// TIA Portal V18 program export: 1 tag tables, 0 data types, 1 data blocks, 7 code blocks (in call order from the OBs), 5 instance data blocks

VAR_GLOBAL   // PLC tag table "Default tag table"
   "Motor start" AT %I0.0 : Bool;
   "Motor Stop" AT %I0.1 : Bool;
   Tag_2 AT %I0.2 : Bool;
   Tag_4 AT %I0.3 : Bool;
   "Motor running LED" AT %Q0.0 : Bool;
   "Motor contactor" AT %Q0.2 : Bool;
   Tag_1 AT %M10.0 : Bool;
   Tag_3 AT %M10.1 : Bool;
   System_Byte AT %MB88 : Byte;
   FirstScan AT %M88.0 : Bool;
   DiagStatusUpdate AT %M88.1 : Bool;
   AlwaysTRUE AT %M88.2 : Bool;
   AlwaysFALSE AT %M88.3 : Bool;
   "System_Byte(1)" AT %MB88 : Byte;
   Clock_Byte AT %MB0 : Byte;
   Clock_10Hz AT %M0.0 : Bool;
   Clock_5Hz AT %M0.1 : Bool;
   "Clock_2.5Hz" AT %M0.2 : Bool;
   Clock_2Hz AT %M0.3 : Bool;
   "Clock_1.25Hz" AT %M0.4 : Bool;
   Clock_1Hz AT %M0.5 : Bool;
   "Clock_0.625Hz" AT %M0.6 : Bool;
   "Clock_0.5Hz" AT %M0.7 : Bool;
   Alarm AT %MW40 : Word;
   Tag_5 AT %M40.0 : Bool;
END_VAR

DATA_BLOCK "Global data"   // DB2
{ S7_Optimized_Access := 'TRUE' }
VERSION : 0.1
// stored: AutoNumber true, DBAccessibleFromOPCUA true, IsOnlyStoredInLoadMemory false, IsRetainMemResEnabled false, IsWriteProtectedInAS false, MemoryReserve 100
   VAR
      data1 : Bool;
      data2 : Bool;
      data3 : Bool;
      data4 : Bool;
      data5 : Bool;
      data6 : Bool;
      data7 : Bool;
      data8 : Bool;
   END_VAR
   VAR RETAIN
      dataB1 : Byte := 10;
   END_VAR
   VAR
      dataB2 : Byte := 10;
      dataB3 : Byte := 10;
      dataB4 : Byte := 10;
      dataW1 : Word := 10;
   END_VAR
   VAR RETAIN
      dataW2 : Word := 20;
      dataW3 : Word := 20;
      dataW4 : Word := 20;
   END_VAR
   VAR
      dataW5 : Word := 20;
   END_VAR
BEGIN
END_DATA_BLOCK

ORGANIZATION_BLOCK "Main"   // OB1, LAD, ProgramCycle
TITLE = "Main Program Sweep (Cycle)"
{ S7_Optimized_Access := 'TRUE' }
VERSION : 0.1
// stored: AutoNumber true, IsIECCheckEnabled false, SetENOAutomatically false
   VAR_INPUT
      Initial_Call : Bool;   // Initial call of this OB
      Remanence : Bool;   // =True, if remanent data are available
   END_VAR
BEGIN

REGION Network 1
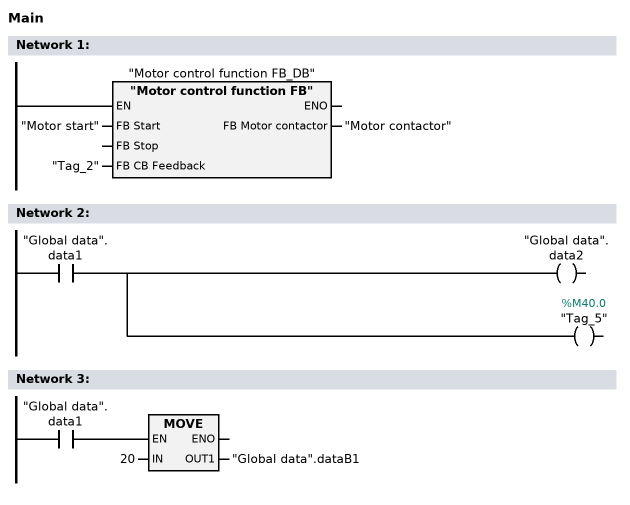
   RUNG wire#powerrail
      "Motor control function FB_DB"("FB Start" := "Motor start", "FB Stop" :=, "FB CB Feedback" := "Tag_2", "FB Motor contactor" => "Motor contactor")
   END_RUNG
   // the same network as SCL:
   "Motor control function FB_DB"("FB Start" := "Motor start",   // "Motor control function FB"
                           "FB CB Feedback" := "Tag_2",
                           "FB Motor contactor" => "Motor contactor");
END_REGION

REGION Network 2
   RUNG wire#powerrail
      Contact( "Global data".data1 )
      wire#w1
      Coil( "Global data".data2 )
   END_RUNG
   RUNG wire#w1
      Coil( "Tag_5" )
   END_RUNG
   // the same network as SCL:
   "Global data".data2 := "Global data".data1;
   "Tag_5" := "Global data".data1;
END_REGION

REGION Network 3
   RUNG wire#powerrail
      Contact( "Global data".data1 )
      Move(in := 20, out1 => "Global data".dataB1)
   END_RUNG
   // the same network as SCL:
   IF "Global data".data1 THEN "Global data".dataB1 := 20; END_IF;
END_REGION
END_ORGANIZATION_BLOCK

FUNCTION_BLOCK "Motor control function FB"   // FB1, LAD
{ S7_Optimized_Access := 'TRUE' }
VERSION : 0.1
// stored: AutoNumber true, IsIECCheckEnabled false, IsRetainMemResEnabled false, MemoryReserve 100, SetENOAutomatically false, UDAEnableTagReadback false
   VAR_INPUT
      "FB Start" : Bool;
      "FB Stop" : Bool;
      "FB CB Feedback" : Bool;
   END_VAR
   VAR_OUTPUT
      "FB Motor contactor" : Bool;
   END_VAR
BEGIN

REGION Network 1: Start motor contactor
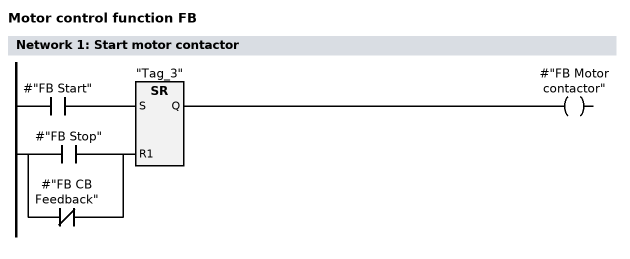
   RUNG wire#powerrail
      Contact( #"FB Start" )
      S_SR(operand := "Tag_3", r1 := wire#w1)
      Coil( #"FB Motor contactor" )
   END_RUNG
   RUNG wire#powerrail
      Contact( #"FB Stop" )
   END_RUNG wire#w1
   RUNG wire#powerrail
      I_Contact( #"FB CB Feedback" )
   END_RUNG wire#w1
   // the same network as SCL:
   IF #"FB Start" THEN
       "Tag_3" := TRUE;   // SR flip-flop
   END_IF;
   IF #"FB Stop" OR NOT #"FB CB Feedback" THEN "Tag_3" := FALSE; END_IF;
   #"FB Motor contactor" := "Tag_3";
END_REGION
END_FUNCTION_BLOCK

FUNCTION "Motor control Function FC" : Void   // FC2, LAD
{ S7_Optimized_Access := 'TRUE' }
VERSION : 0.1
// stored: AutoNumber true, IsIECCheckEnabled false, SetENOAutomatically false, UDAEnableTagReadback false
   VAR_INPUT
      Start : Bool;   // Input to start motor
      Stop : Bool;   // input to stop motor
      "CB feedback" : Bool;
   END_VAR
   VAR_OUTPUT
      "Motor contactor" : Bool;   // Start motor contactor
   END_VAR
BEGIN

REGION Network 1: Start motor contactor
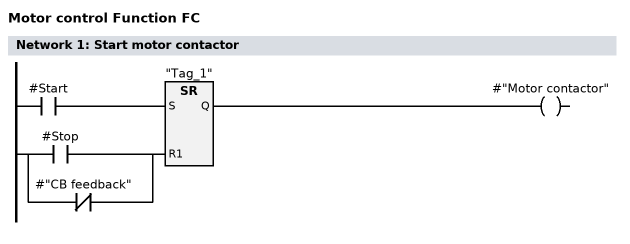
   RUNG wire#powerrail
      Contact( #Start )
      S_SR(operand := "Tag_1", r1 := wire#w1)
      Coil( #"Motor contactor" )
   END_RUNG
   RUNG wire#powerrail
      Contact( #Stop )
   END_RUNG wire#w1
   RUNG wire#powerrail
      I_Contact( #"CB feedback" )
   END_RUNG wire#w1
   // the same network as SCL:
   IF #Start THEN
       "Tag_1" := TRUE;   // SR flip-flop
   END_IF;
   IF #Stop OR NOT #"CB feedback" THEN "Tag_1" := FALSE; END_IF;
   #"Motor contactor" := "Tag_1";
END_REGION
END_FUNCTION

FUNCTION "Motor_control_FC" : Void   // FC1, LAD
{ S7_Optimized_Access := 'TRUE' }
VERSION : 0.1
// stored: AutoNumber true, IsIECCheckEnabled false, SetENOAutomatically false, UDAEnableTagReadback false
BEGIN

REGION Network 1
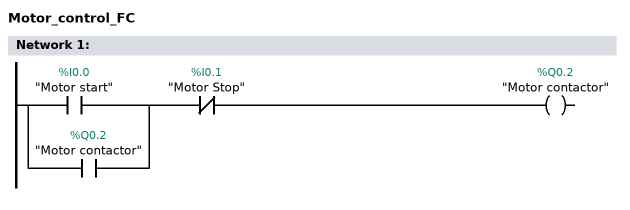
   RUNG wire#powerrail
      Contact( "Motor start" )
      wire#w1
      I_Contact( "Motor Stop" )
      Coil( "Motor contactor" )
   END_RUNG
   RUNG wire#powerrail
      Contact( "Motor contactor" )
   END_RUNG wire#w1
   // the same network as SCL:
   "Motor contactor" := ("Motor start" OR "Motor contactor") AND NOT "Motor Stop";
END_REGION
END_FUNCTION

FUNCTION_BLOCK "Multi instance FB"   // FB2, LAD
{ S7_Optimized_Access := 'TRUE' }
VERSION : 0.1
// stored: AutoNumber true, IsIECCheckEnabled false, IsRetainMemResEnabled false, MemoryReserve 100, SetENOAutomatically false, UDAEnableTagReadback false
   VAR
      "Motor control function FB_Instance" { S7_SetPoint := 'True'} : "Motor control function FB";
      "Motor control function FB_Instance_1" { S7_SetPoint := 'True'} : "Motor control function FB";
   END_VAR
BEGIN

REGION Network 1: Motor 1
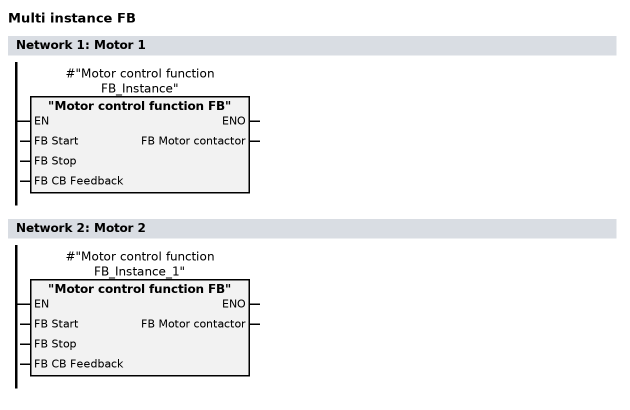
   RUNG wire#powerrail
      #"Motor control function FB_Instance"("FB Start" :=, "FB Stop" :=, "FB CB Feedback" :=, "FB Motor contactor" =>)
   END_RUNG
   // the same network as SCL:
   #"Motor control function FB_Instance"();   // "Motor control function FB"
END_REGION

REGION Network 2: Motor 2
   RUNG wire#powerrail
      #"Motor control function FB_Instance_1"("FB Start" :=, "FB Stop" :=, "FB CB Feedback" :=, "FB Motor contactor" =>)
   END_RUNG
   // the same network as SCL:
   #"Motor control function FB_Instance_1"();   // "Motor control function FB"
END_REGION
END_FUNCTION_BLOCK

FUNCTION "Sunc_2" : Void   // FC4, LAD
{ S7_Optimized_Access := 'TRUE' }
VERSION : 0.1
// stored: AutoNumber true, IsIECCheckEnabled false, SetENOAutomatically false, UDAEnableTagReadback false
BEGIN

REGION Network 1
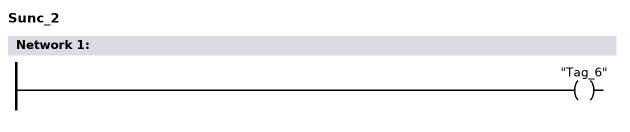
   RUNG wire#powerrail
      Coil( "Tag_6" )
   END_RUNG
   // the same network as SCL:
   "Tag_6" := TRUE;
END_REGION
END_FUNCTION

FUNCTION "Sync_Test" : Void   // FC3, LAD
{ S7_Optimized_Access := 'TRUE' }
VERSION : 0.1
// stored: AutoNumber true, IsIECCheckEnabled false, SetENOAutomatically false, UDAEnableTagReadback false
BEGIN

REGION Network 1
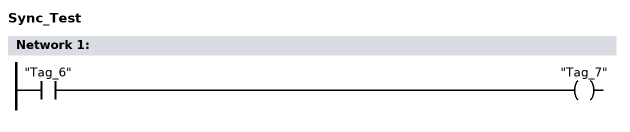
   RUNG wire#powerrail
      Contact( "Tag_6" )
      Coil( "Tag_7" )
   END_RUNG
   // the same network as SCL:
   "Tag_7" := "Tag_6";
END_REGION
END_FUNCTION

DATA_BLOCK "Motor control function FB_DB"   // DB1
VERSION : 0.1
// stored: AutoNumber true, DBAccessibleFromOPCUA true, InstanceOfName Motor control function FB, InstanceOfType FB
"Motor control function FB"
BEGIN
END_DATA_BLOCK

DATA_BLOCK "Motor control function FB_DB_1"   // DB3
VERSION : 0.1
// stored: AutoNumber true, DBAccessibleFromOPCUA true, InstanceOfName Motor control function FB, InstanceOfType FB
"Motor control function FB"
BEGIN
END_DATA_BLOCK

DATA_BLOCK "Motor control function FB_DB_2"   // DB5
VERSION : 0.1
// stored: AutoNumber true, DBAccessibleFromOPCUA true, InstanceOfName Motor control function FB, InstanceOfType FB
"Motor control function FB"
BEGIN
END_DATA_BLOCK

DATA_BLOCK "Multi instance FB_DB"   // DB4
VERSION : 0.1
// stored: AutoNumber true, DBAccessibleFromOPCUA true, InstanceOfName Multi instance FB, InstanceOfType FB
"Multi instance FB"
BEGIN
END_DATA_BLOCK

DATA_BLOCK "Multi instance FB_DB_1"   // DB6
VERSION : 0.1
// stored: AutoNumber true, DBAccessibleFromOPCUA true, InstanceOfName Multi instance FB, InstanceOfType FB
"Multi instance FB"
BEGIN
END_DATA_BLOCK
